# EPICS autosave request: iocBoot/sioc-esb-tps03/tps.req
file ../tpsCommon.req P=$(P)
